(* PLC project MotorControlProject, Example Corp MotorController 1.0, author Engineer *)
(* stored: creationDateTime 2024-03-15 10:30:00, organization Example Corp, modificationDateTime 2024-03-15 14:22:00, version 1.0 *)

PROGRAM MotorControl
  VAR
    MotorSpeed : INT;
    IsRunning : BOOL;
  END_VAR

            
IF IsRunning THEN
    MotorSpeed := 100;
ELSE
    MotorSpeed := 0;
END_IF;
            
          
END_PROGRAM

CONFIGURATION Config0
  RESOURCE Res0 ON PLC
    TASK Task0(INTERVAL := T#20ms, PRIORITY := 0);
    PROGRAM MotorControl0 WITH Task0 : MotorControl;
  END_RESOURCE
END_CONFIGURATION
